DATA_BLOCK "IEC_Timer_CylRetract"
{ S7_Optimized_Access := 'TRUE' }
VERSION : 0.1
NON_RETAIN
IEC_TIMER
BEGIN
END_DATA_BLOCK
